# B&R Automation Studio project Lektion_10_agdp
Automation Studio 4.8.2.72

## Configuration Config1

### Task classes (Cpu.sw)
```
Cyclic#4:
  Assignment <- Assignment1.prg
  Assignmen1 <- Assignment2.prg
Binaries: udbdef, FWRules, TCData, sysconf, Role, User, iomap, ashwd, asfw, arconfig, ashwac
Libraries: AsTCP, runtime, AsBrStr, astime, asieccon
```

### Hardware
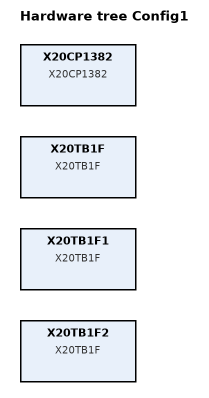
```
X20CP1382 : X20CP1382 v1.10.0.0  [X1 -> X1.SL; X2 -> X2.SL; X3 -> X3.SL]
  Module X1 (Type=X1, Virtual=true, Version=1.10.0.0)
    Connection (Connector=SS1, TargetModule=X20TB1F, TargetConnector=SS)
    Connection (Connector=SL, TargetModule=X20CP1382, TargetConnector=X1)
  Module X2 (Type=X2, Virtual=true, Version=1.10.0.0)
    Connection (Connector=SS1, TargetModule=X20TB1F1, TargetConnector=SS)
    Connection (Connector=SL, TargetModule=X20CP1382, TargetConnector=X2)
  Module X3 (Type=X3, Virtual=true, Version=1.10.0.0)
    Connection (Connector=SS1, TargetModule=X20TB1F2, TargetConnector=SS)
    Connection (Connector=SL, TargetModule=X20CP1382, TargetConnector=X3)
  Connector IF2:
    ActivateDevice = 1
  ConfigurationID = Lektion_10_agdp_Config1
  Simulation = 1
X20TB1F : X20TB1F v1.0.0.0
X20TB1F1 : X20TB1F v1.0.0.0
X20TB1F2 : X20TB1F v1.0.0.0
```

## Logical view

Binary libraries used (declarations not repeated): operator, runtime, astime, AsIecCon, AsTCP, AsBrStr

### Program Logical/Assignment1

#### Main.st
```iecst
PROGRAM _INIT
	tcpst := TCPSTATE_SOCKET_OPEN;
END_PROGRAM

PROGRAM _CYCLIC
	CASE tcpst OF
		TCPSTATE_SOCKET_OPEN :
			TcpOpen1.enable := TRUE;
			TcpOpen1.port := 12345;
			TcpOpen1.options := tcpOPT_REUSEADDR;
			TcpOpen1();
			IF (TcpOpen1.status = ERR_OK) THEN
				tcpst := TCPSTATE_SERVER_CREATE;
			END_IF

		TCPSTATE_SERVER_CREATE :
			TcpServer1.enable := TRUE;
			TcpServer1.ident := TcpOpen1.ident;
			TcpServer1();
			IF (TcpServer1.status = ERR_OK) THEN
				tcpst := TCPSTATE_RECEIVE;
				receiveData := DELETE(receiveData, LEN(receiveData), 1); // Ny kode
			END_IF

		TCPSTATE_RECEIVE :
			TcpReceive1.enable := TRUE;
			TcpReceive1.ident := TcpServer1.identclnt;
			TcpReceive1.pData := ADR(receiveData);
			TcpReceive1.datamax := SIZEOF(receiveData);
			TcpReceive1();
			IF (TcpReceive1.status = ERR_OK) THEN
				tcpst := TCPSTATE_SEND;
				sendData := receiveData;
			END_IF

		TCPSTATE_SEND :
			TcpSend1.enable := TRUE;
			TcpSend1.ident := TcpServer1.identclnt;
			TcpSend1.pData := ADR(sendData);
			TcpSend1.datalen := brsstrlen(ADR(sendData));     // We use brsstrlen() to get the length in UDINT datatype
			TcpSend1();
			IF (TcpSend1.status = ERR_OK) THEN
				tcpst := TCPSTATE_CLOSE;
			END_IF

		TCPSTATE_CLOSE :
			sendData := receiveData := '';
			TcpClose1.enable := TRUE;
			TcpClose1.ident := TcpServer1.identclnt;
			TcpClose1();
			IF (TcpClose1.status = ERR_OK) THEN
				TcpServer1.enable := FALSE;
				TcpServer1();
				tcpst := TCPSTATE_SERVER_CREATE;
			END_IF

	END_CASE

END_PROGRAM

PROGRAM _EXIT
	TcpClose1.enable := TRUE;
	TcpClose1.ident := TcpServer1.identclnt;
	TcpClose1();

	TcpClose2.enable := TRUE;
	TcpClose2.ident := TcpOpen1.ident;
	TcpClose2();

END_PROGRAM
```

### Types.typ
```iecst
TYPE
	TCPSTATE :
		(
		TCPSTATE_SOCKET_OPEN,
		TCPSTATE_SERVER_CREATE,
		TCPSTATE_RECEIVE,
		TCPSTATE_SEND,
		TCPSTATE_CLOSE
	);
END_TYPE
```

### Program Logical/Program

#### Variables.var
```iecst
VAR
	tcpst : TCPSTATE;
	sendData : STRING[80];
	receiveData : STRING[80];
	TcpOpen1 : TcpOpen;
	TcpServer1 : TcpServer;
	TcpReceive1 : TcpRecv;
	TcpSend1 : TcpSend;
	TcpClose1 : TcpClose;
	TcpClose2 : TcpClose;
	testUA : INT;
	saver : STRING[80];
END_VAR
```

#### Main.st
```iecst
PROGRAM _INIT
	tcpst := TCPSTATE_SOCKET_OPEN;
END_PROGRAM

PROGRAM _CYCLIC
	CASE tcpst OF
		TCPSTATE_SOCKET_OPEN :
			TcpOpen1.enable := TRUE;
			TcpOpen1.port := 12345;
			TcpOpen1.options := tcpOPT_REUSEADDR;
			TcpOpen1();
			IF (TcpOpen1.status = ERR_OK) THEN
				tcpst := TCPSTATE_SERVER_CREATE;
			END_IF

		TCPSTATE_SERVER_CREATE :
			TcpServer1.enable := TRUE;
			TcpServer1.ident := TcpOpen1.ident;
			TcpServer1();
			IF (TcpServer1.status = ERR_OK) THEN
				tcpst := TCPSTATE_RECEIVE;
			END_IF

		TCPSTATE_RECEIVE :
			TcpReceive1.enable := TRUE;
			TcpReceive1.ident := TcpServer1.identclnt;
			TcpReceive1.pData := ADR(receiveData);
			TcpReceive1.datamax := SIZEOF(receiveData);
			TcpReceive1();
			IF (TcpReceive1.status = ERR_OK) THEN
				saver := '';
				saver := receiveData;
				tcpst := TCPSTATE_SEND;
				sendData := receiveData;
				TcpReceive1.datamax := SIZEOF('');
			END_IF

		TCPSTATE_SEND :
			TcpSend1.enable := TRUE;
			TcpSend1.ident := TcpServer1.identclnt;
			TcpSend1.pData := ADR(sendData);
			TcpSend1.datalen := brsstrlen(ADR(sendData));     // We use brsstrlen() to get the length in UDINT datatype
			TcpSend1();
			IF (TcpSend1.status = ERR_OK) THEN
				tcpst := TCPSTATE_CLOSE;
			END_IF

		TCPSTATE_CLOSE :
			sendData := receiveData := '';
			TcpClose1.enable := TRUE;
			TcpClose1.ident := TcpServer1.identclnt;
			TcpClose1();
			IF (TcpClose1.status = ERR_OK) THEN
				TcpServer1.enable := FALSE;
				TcpServer1();
				tcpst := TCPSTATE_SERVER_CREATE;
			END_IF

	END_CASE

END_PROGRAM

PROGRAM _EXIT
	TcpClose1.enable := TRUE;
	TcpClose1.ident := TcpServer1.identclnt;
	TcpClose1();

	TcpClose2.enable := TRUE;
	TcpClose2.ident := TcpOpen1.ident;
	TcpClose2();

END_PROGRAM
```
